// Mitsubishi GX Works2 project: Melsec   PLC: FX3U/FX3UC

PROGRAM MAIN
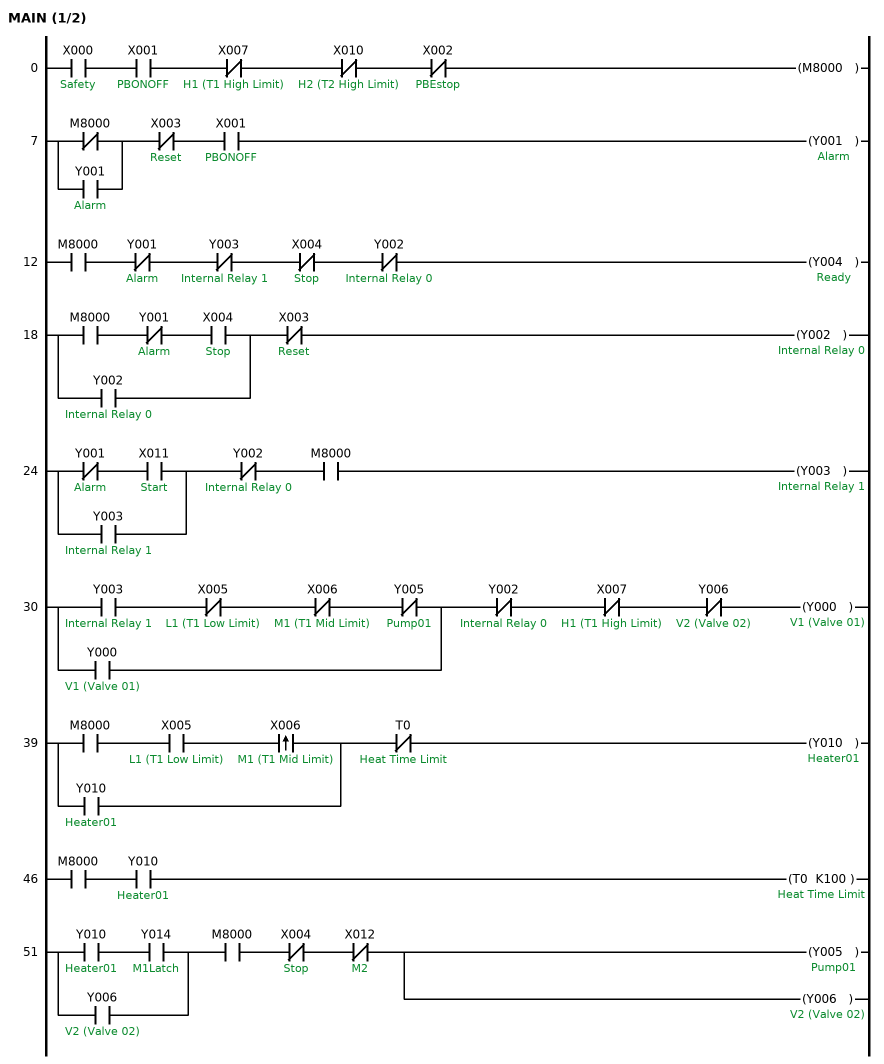
0     LD      X000  ; Safety
      AND     X001  ; PBONOFF
      ANI     X007  ; H1 (T1 High Limit)
      ANI     X010  ; H2 (T2 High Limit)
      ANI     X002  ; PBEstop
      OUT     M8000
7     LDI     M8000
      OR      Y001  ; Alarm
      ANI     X003  ; Reset
      AND     X001  ; PBONOFF
      OUT     Y001  ; Alarm
12    LD      M8000
      ANI     Y001  ; Alarm
      ANI     Y003  ; Internal Relay 1
      ANI     X004  ; Stop
      ANI     Y002  ; Internal Relay 0
      OUT     Y004  ; Ready
18    LD      M8000
      ANI     Y001  ; Alarm
      AND     X004  ; Stop
      OR      Y002  ; Internal Relay 0
      ANI     X003  ; Reset
      OUT     Y002  ; Internal Relay 0
24    LDI     Y001  ; Alarm
      AND     X011  ; Start
      OR      Y003  ; Internal Relay 1
      ANI     Y002  ; Internal Relay 0
      AND     M8000
      OUT     Y003  ; Internal Relay 1
30    LD      Y003  ; Internal Relay 1
      ANI     X005  ; L1 (T1 Low Limit)
      ANI     X006  ; M1 (T1 Mid Limit)
      ANI     Y005  ; Pump01
      OR      Y000  ; V1 (Valve 01)
      ANI     Y002  ; Internal Relay 0
      ANI     X007  ; H1 (T1 High Limit)
      ANI     Y006  ; V2 (Valve 02)
      OUT     Y000  ; V1 (Valve 01)
39    LD      M8000
      AND     X005  ; L1 (T1 Low Limit)
      ANDP    X006  ; M1 (T1 Mid Limit)
      OR      Y010  ; Heater01
      ANI     T0  ; Heat Time Limit
      OUT     Y010  ; Heater01
46    LD      M8000
      AND     Y010  ; Heater01
      OUT     T0 K100  ; Heat Time Limit
51    LD      Y010  ; Heater01
      AND     Y014  ; M1Latch
      OR      Y006  ; V2 (Valve 02)
      AND     M8000
      ANI     X004  ; Stop
      ANI     X012  ; M2
      OUT     Y005  ; Pump01
      OUT     Y006  ; V2 (Valve 02)
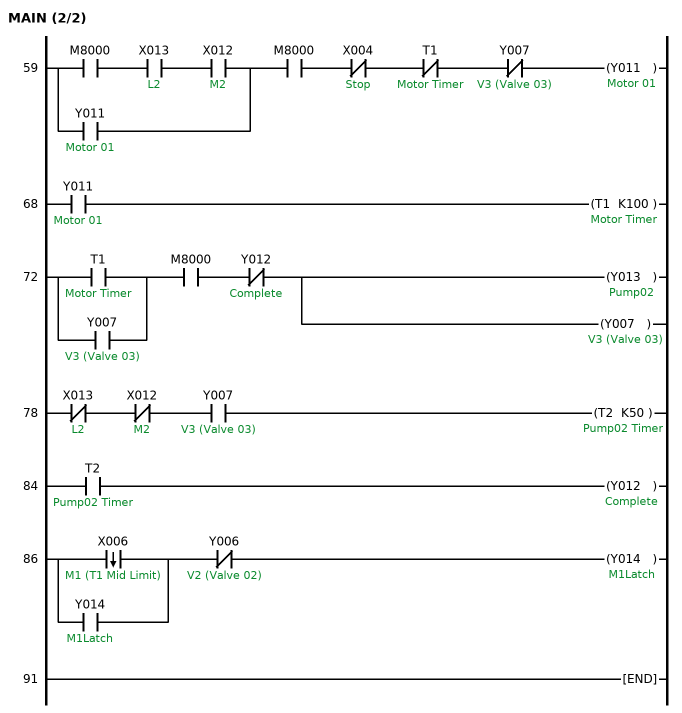
59    LD      M8000
      AND     X013  ; L2
      AND     X012  ; M2
      OR      Y011  ; Motor 01
      AND     M8000
      ANI     X004  ; Stop
      ANI     T1  ; Motor Timer
      ANI     Y007  ; V3 (Valve 03)
      OUT     Y011  ; Motor 01
68    LD      Y011  ; Motor 01
      OUT     T1 K100  ; Motor Timer
72    LD      T1  ; Motor Timer
      OR      Y007  ; V3 (Valve 03)
      AND     M8000
      ANI     Y012  ; Complete
      OUT     Y013  ; Pump02
      OUT     Y007  ; V3 (Valve 03)
78    LDI     X013  ; L2
      ANI     X012  ; M2
      AND     Y007  ; V3 (Valve 03)
      OUT     T2 K50  ; Pump02 Timer
84    LD      T2  ; Pump02 Timer
      OUT     Y012  ; Complete
86    LDF     X006  ; M1 (T1 Mid Limit)
      OR      Y014  ; M1Latch
      ANI     Y006  ; V2 (Valve 02)
      OUT     Y014  ; M1Latch
91    END
END_PROGRAM

// device comments not shown above
M4000  ; Internal Safety Relay
